(* IEC 61131-3 sources: OpenPLC_Sample_Programs/successed_ST (part 7) *)

(* ---- Scenario7v1_Final.xml_Main.st ---- *)
TYPE
    Magazin_states_t : (Green_Lamp , Init , Interstep , Magazin_Init , Magazin_Init_2 , Slider_Move_Back , Start_Magazin , Step0 , Step1 , convey);
    Stamp_states_t : (Green_Lamp , Init , Interstep , Interstep_2 , StampProcess , StampSliderBack , StampSliderForward , Stamp_Init_1 , Stamp_Init_2 , Stamp_Init_3 , Stamp_Init_4 , Start_Stamp , Step0 , Step1 , Step2);
    Crane_states_t : (Crane_Go_Up , Crane_Init , Crane_Init_2 , Crane_Lift_At_Stamp , Crane_Lift_At_Stamp2 , Crane_Lift_Conveyor , Crane_Lift_Conveyor2 , Crane_Lift_Conveyor_Black , Crane_Lift_Magazin , Crane_Lift_Magazin_Metallic , Crane_Lift_NOT_Metallic_Black , Crane_Lower , Crane_On_Conveyor , Crane_On_Conveyor_Metallic , Crane_On_Conveyor_Metallic2 , Crane_On_Conveyor_Not_Metallica_Black , Crane_On_Stamp_Metallic , Crane_On_Stamp_Metallic2 , Crane_On_Stamp_Metallic2_Lower , Crane_On_Stamp_Stop_Black , Crane_Turn_Left_Back_To_Stamp , Crane_Turn_Left_From_Stamp , Crane_Turn_Left_Metallic , Crane_Turn_Left_Metallic2 , Crane_Turn_Left_NOT_Metallic , Crane_Turn_Left_NOT_Metallic_Black , Crane_Turn_Right_From_Stamp , Init , Interstep , Interstep_2 , Interstep_4 , Lower_Crane , Magazin_Stop , Magazin_Stop_Black , Magazin_Stop_Final , No_Workpiece_ready , Reset_interconnect , Start_Crane , Step0 , Step4 , Suck_At_Stamp , Suck_At_Stamp2 , TimeDelay , Turn_Right , Turn_Right_Black , Turn_Right_Final , pause , release , release2 , release_Black , release_Workpiece);
END_TYPE

FUNCTION_BLOCK Crane_FB
    VAR_INPUT  CraneDown : BOOL; END_VAR
    VAR_OUTPUT  CraneLower : BOOL; END_VAR
    VAR_INPUT  CraneOnConveyor : BOOL; END_VAR
    VAR_INPUT  CraneOnMagazin : BOOL; END_VAR
    VAR_INPUT  CranePositionStamp : BOOL; END_VAR
    VAR_INPUT  CraneSucked : BOOL; END_VAR
    VAR_OUTPUT  CraneTurnClockwise : BOOL; END_VAR
    VAR_OUTPUT  CraneTurnCounterclockwise : BOOL; END_VAR
    VAR_INPUT  CraneUp : BOOL; END_VAR
    VAR  Duration1 : TIME := TIME#1s500ms; END_VAR
    VAR_INPUT  MagazinCapacitiveSensor : BOOL; END_VAR
    VAR_INPUT  MagazinOpticalSensor : BOOL; END_VAR
    VAR_OUTPUT  MagazinVacuumOff : BOOL; END_VAR
    VAR_OUTPUT  MagazinVacuumOn : BOOL; END_VAR
    VAR  SFCInit : BOOL; END_VAR
    VAR_INPUT  SFCReset : BOOL; END_VAR
    VAR_INPUT  SliderMovedOut : BOOL; END_VAR
    VAR_INPUT  SliderNotMovedOut : BOOL; END_VAR
    VAR_INPUT  StampLowered : BOOL; END_VAR
    VAR_INPUT  StampSliderFilled : BOOL; END_VAR
    VAR_INPUT  StampSliderSensorMovedOut : BOOL; END_VAR
    VAR_INPUT  StartButtonMagazin : BOOL; END_VAR
    VAR_OUTPUT  StartCommandCrane : BOOL; END_VAR
    VAR_INPUT  StartVar : BOOL; END_VAR
    VAR  TimeDelay_Timer : TON; END_VAR
    VAR  TimeDelay_Timer_Duration : TIME := TIME#50ms; END_VAR
    VAR  TimeDelay_Timer_interconnect : BOOL; END_VAR
    VAR  Timer1 : TON; END_VAR
    VAR_INPUT  WorkpieceReady : BOOL; END_VAR
    VAR  _state : Crane_states_t; END_VAR
    VAR  _transit : BOOL; END_VAR
    VAR  actualtime1 : TIME; END_VAR
    VAR  interconnect : BOOL; END_VAR
    VAR  interconnectCraneStartCommand : BOOL; END_VAR

    CASE _state OF
        Crane_states_t#Crane_Go_Up:
            _transit := FALSE;
            CraneLower := FALSE;
            IF ((CraneUp AND WorkpieceReady) AND (NOT MagazinCapacitiveSensor AND NOT MagazinOpticalSensor)) THEN
                _transit := TRUE;
                _state := Crane_states_t#Turn_Right_Black;
            ELSIF ((CraneUp AND WorkpieceReady) AND (MagazinCapacitiveSensor OR MagazinOpticalSensor)) THEN
                _transit := TRUE;
                _state := Crane_states_t#pause;
            ELSIF (CraneUp AND NOT WorkpieceReady) THEN
                _transit := TRUE;
                _state := Crane_states_t#Step4;
            END_IF;

        Crane_states_t#Crane_Init:
            _transit := FALSE;
            CraneLower := TRUE;
            interconnectCraneStartCommand := FALSE;
            IF CraneDown THEN
                _transit := TRUE;
                _state := Crane_states_t#Crane_Init_2;
            END_IF;

        Crane_states_t#Crane_Init_2:
            _transit := FALSE;
            CraneLower := FALSE;
            IF CraneUp THEN
                _transit := TRUE;
                _state := Crane_states_t#Interstep;
            END_IF;

        Crane_states_t#Crane_Lift_At_Stamp:
            _transit := FALSE;
            CraneLower := FALSE;
            IF CraneUp THEN
                _transit := TRUE;
                _state := Crane_states_t#Crane_Turn_Left_From_Stamp;
            END_IF;

        Crane_states_t#Crane_Lift_At_Stamp2:
            _transit := FALSE;
            CraneLower := FALSE;
            IF CraneUp THEN
                _transit := TRUE;
                _state := Crane_states_t#Crane_Turn_Right_From_Stamp;
            END_IF;

        Crane_states_t#Crane_Lift_Conveyor:
            _transit := FALSE;
            CraneLower := FALSE;
            IF TRUE THEN
                _transit := TRUE;
                _state := Crane_states_t#Interstep;
            END_IF;

        Crane_states_t#Crane_Lift_Conveyor2:
            _transit := FALSE;
            CraneLower := FALSE;
            IF TRUE THEN
                _transit := TRUE;
                _state := Crane_states_t#Interstep;
            END_IF;

        Crane_states_t#Crane_Lift_Conveyor_Black:
            _transit := FALSE;
            CraneLower := FALSE;
            IF CraneUp THEN
                _transit := TRUE;
                _state := Crane_states_t#Crane_Turn_Left_Back_To_Stamp;
            END_IF;

        Crane_states_t#Crane_Lift_Magazin:
            _transit := FALSE;
            CraneLower := FALSE;
            IF CraneUp THEN
                _transit := TRUE;
                _state := Crane_states_t#Crane_Turn_Left_NOT_Metallic;
            END_IF;

        Crane_states_t#Crane_Lift_Magazin_Metallic:
            _transit := FALSE;
            CraneLower := FALSE;
            IF CraneUp THEN
                _transit := TRUE;
                _state := Crane_states_t#Crane_Turn_Left_Metallic;
            END_IF;

        Crane_states_t#Crane_Lift_NOT_Metallic_Black:
            _transit := FALSE;
            CraneLower := FALSE;
            IF CraneUp THEN
                _transit := TRUE;
                _state := Crane_states_t#Crane_Turn_Left_NOT_Metallic_Black;
            END_IF;

        Crane_states_t#Crane_Lower:
            _transit := FALSE;
            MagazinVacuumOn := TRUE;
            MagazinVacuumOff := FALSE;
            CraneLower := TRUE;
            IF CraneSucked THEN
                _transit := TRUE;
                _state := Crane_states_t#Step0;
            END_IF;

        Crane_states_t#Crane_On_Conveyor:
            _transit := FALSE;
            CraneTurnCounterclockwise := FALSE;
            CraneTurnClockwise := FALSE;
            CraneLower := TRUE;
            IF CraneDown THEN
                _transit := TRUE;
                _state := Crane_states_t#release;
            END_IF;

        Crane_states_t#Crane_On_Conveyor_Metallic:
            _transit := FALSE;
            CraneTurnCounterclockwise := FALSE;
            CraneTurnClockwise := FALSE;
            CraneLower := TRUE;
            IF CraneDown THEN
                _transit := TRUE;
                _state := Crane_states_t#release;
            END_IF;

        Crane_states_t#Crane_On_Conveyor_Metallic2:
            _transit := FALSE;
            CraneTurnCounterclockwise := FALSE;
            CraneTurnClockwise := FALSE;
            CraneLower := TRUE;
            IF CraneDown THEN
                _transit := TRUE;
                _state := Crane_states_t#release2;
            END_IF;

        Crane_states_t#Crane_On_Conveyor_Not_Metallica_Black:
            _transit := FALSE;
            CraneTurnCounterclockwise := FALSE;
            CraneTurnClockwise := FALSE;
            CraneLower := TRUE;
            IF CraneDown THEN
                _transit := TRUE;
                _state := Crane_states_t#release_Black;
            END_IF;

        Crane_states_t#Crane_On_Stamp_Metallic:
            _transit := FALSE;
            CraneTurnCounterclockwise := FALSE;
            CraneTurnClockwise := FALSE;
            CraneLower := TRUE;
            IF CraneDown THEN
                _transit := TRUE;
                _state := Crane_states_t#release_Workpiece;
            END_IF;

        Crane_states_t#Crane_On_Stamp_Metallic2:
            _transit := FALSE;
            CraneTurnCounterclockwise := FALSE;
            CraneTurnClockwise := FALSE;
            IF StampLowered THEN
                _transit := TRUE;
                _state := Crane_states_t#Interstep_4;
            END_IF;

        Crane_states_t#Crane_On_Stamp_Metallic2_Lower:
            _transit := FALSE;
            CraneLower := TRUE;
            IF CraneDown THEN
                _transit := TRUE;
                _state := Crane_states_t#Suck_At_Stamp2;
            END_IF;

        Crane_states_t#Crane_On_Stamp_Stop_Black:
            _transit := FALSE;
            CraneTurnClockwise := FALSE;
            CraneTurnCounterclockwise := FALSE;
            IF TRUE THEN
                _transit := TRUE;
                _state := Crane_states_t#Reset_interconnect;
            END_IF;

        Crane_states_t#Crane_Turn_Left_Back_To_Stamp:
            _transit := FALSE;
            CraneTurnCounterclockwise := TRUE;
            CraneTurnClockwise := FALSE;
            IF CranePositionStamp THEN
                _transit := TRUE;
                _state := Crane_states_t#Crane_On_Stamp_Stop_Black;
            END_IF;

        Crane_states_t#Crane_Turn_Left_From_Stamp:
            _transit := FALSE;
            CraneTurnClockwise := TRUE;
            CraneTurnCounterclockwise := FALSE;
            IF CraneOnConveyor THEN
                _transit := TRUE;
                _state := Crane_states_t#Crane_On_Conveyor_Metallic;
            END_IF;

        Crane_states_t#Crane_Turn_Left_Metallic:
            _transit := FALSE;
            CraneTurnCounterclockwise := TRUE;
            CraneTurnClockwise := FALSE;
            IF CranePositionStamp THEN
                _transit := TRUE;
                _state := Crane_states_t#Crane_On_Stamp_Metallic;
            END_IF;

        Crane_states_t#Crane_Turn_Left_Metallic2:
            _transit := FALSE;
            CraneTurnCounterclockwise := TRUE;
            CraneTurnClockwise := FALSE;
            IF CranePositionStamp THEN
                _transit := TRUE;
                _state := Crane_states_t#Crane_On_Stamp_Metallic2;
            END_IF;

        Crane_states_t#Crane_Turn_Left_NOT_Metallic:
            _transit := FALSE;
            CraneTurnCounterclockwise := TRUE;
            CraneTurnClockwise := FALSE;
            IF CraneOnConveyor THEN
                _transit := TRUE;
                _state := Crane_states_t#Crane_On_Conveyor;
            END_IF;

        Crane_states_t#Crane_Turn_Left_NOT_Metallic_Black:
            _transit := FALSE;
            CraneTurnCounterclockwise := TRUE;
            CraneTurnClockwise := FALSE;
            IF CraneOnConveyor THEN
                _transit := TRUE;
                _state := Crane_states_t#Crane_On_Conveyor_Not_Metallica_Black;
            END_IF;

        Crane_states_t#Crane_Turn_Right_From_Stamp:
            _transit := FALSE;
            CraneTurnClockwise := TRUE;
            CraneTurnCounterclockwise := FALSE;
            IF CraneOnConveyor THEN
                _transit := TRUE;
                _state := Crane_states_t#Crane_On_Conveyor_Metallic2;
            END_IF;

        Crane_states_t#Init:
            _transit := FALSE;
            IF TRUE THEN
                _transit := TRUE;
                _state := Crane_states_t#Start_Crane;
            END_IF;

        Crane_states_t#Interstep:
            _transit := FALSE;
            StartCommandCrane := TRUE;
            IF StartVar THEN
                _transit := TRUE;
                _state := Crane_states_t#Interstep_2;
            END_IF;

        Crane_states_t#Interstep_2:
            _transit := FALSE;
            IF SliderMovedOut THEN
                _transit := TRUE;
                _state := Crane_states_t#TimeDelay;
            END_IF;

        Crane_states_t#Interstep_4:
            _transit := FALSE;
            IF StampSliderSensorMovedOut THEN
                _transit := TRUE;
                _state := Crane_states_t#Crane_On_Stamp_Metallic2_Lower;
            END_IF;

        Crane_states_t#Lower_Crane:
            _transit := FALSE;
            CraneLower := TRUE;
            IF CraneDown THEN
                _transit := TRUE;
                _state := Crane_states_t#Suck_At_Stamp;
            END_IF;

        Crane_states_t#Magazin_Stop:
            _transit := FALSE;
            CraneTurnClockwise := FALSE;
            CraneTurnCounterclockwise := FALSE;
            IF TRUE THEN
                _transit := TRUE;
                _state := Crane_states_t#Crane_Lower;
            END_IF;

        Crane_states_t#Magazin_Stop_Black:
            _transit := FALSE;
            CraneTurnClockwise := FALSE;
            CraneTurnCounterclockwise := FALSE;
            MagazinVacuumOn := TRUE;
            MagazinVacuumOff := FALSE;
            CraneLower := TRUE;
            IF CraneSucked THEN
                _transit := TRUE;
                _state := Crane_states_t#Crane_Lift_NOT_Metallic_Black;
            END_IF;

        Crane_states_t#Magazin_Stop_Final:
            _transit := FALSE;
            CraneTurnClockwise := FALSE;
            CraneTurnCounterclockwise := FALSE;
            IF TRUE THEN
                _transit := TRUE;
                _state := Crane_states_t#Start_Crane;
            END_IF;

        Crane_states_t#No_Workpiece_ready:
            _transit := FALSE;
            MagazinVacuumOn := FALSE;
            MagazinVacuumOff := FALSE;
            CraneLower := FALSE;
            IF NOT StampSliderFilled THEN
                _transit := TRUE;
                _state := Crane_states_t#Turn_Right_Final;
            ELSIF StampSliderFilled THEN
                _transit := TRUE;
                _state := Crane_states_t#Crane_Turn_Left_Metallic2;
            END_IF;

        Crane_states_t#Reset_interconnect:
            _transit := FALSE;
            interconnect := FALSE;
            Timer1(IN := FALSE, PT := TIME#1ms);
            IF SliderMovedOut THEN
                _transit := TRUE;
                _state := Crane_states_t#Lower_Crane;
            END_IF;

        Crane_states_t#Start_Crane:
            _transit := FALSE;
            CraneLower := FALSE;
            MagazinVacuumOff := FALSE;
            MagazinVacuumOn := FALSE;
            CraneTurnCounterclockwise := FALSE;
            CraneTurnClockwise := FALSE;
            StartVar := FALSE;
            StartCommandCrane := FALSE;
            IF (StartButtonMagazin = TRUE) THEN
                interconnectCraneStartCommand := TRUE;
            END_IF;
            IF interconnectCraneStartCommand THEN
                _transit := TRUE;
                _state := Crane_states_t#Crane_Init;
            END_IF;

        Crane_states_t#Step0:
            _transit := FALSE;
            IF (MagazinCapacitiveSensor OR MagazinOpticalSensor) THEN
                _transit := TRUE;
                _state := Crane_states_t#Crane_Lift_Magazin_Metallic;
            ELSIF (NOT MagazinCapacitiveSensor AND NOT MagazinOpticalSensor) THEN
                _transit := TRUE;
                _state := Crane_states_t#Crane_Lift_Magazin;
            END_IF;

        Crane_states_t#Step4:
            _transit := FALSE;
            IF TRUE THEN
                _transit := TRUE;
                _state := Crane_states_t#Interstep;
            END_IF;

        Crane_states_t#Suck_At_Stamp:
            _transit := FALSE;
            MagazinVacuumOn := TRUE;
            MagazinVacuumOff := FALSE;
            IF CraneSucked THEN
                _transit := TRUE;
                _state := Crane_states_t#Crane_Lift_At_Stamp;
            END_IF;

        Crane_states_t#Suck_At_Stamp2:
            _transit := FALSE;
            MagazinVacuumOn := TRUE;
            MagazinVacuumOff := FALSE;
            IF CraneSucked THEN
                _transit := TRUE;
                _state := Crane_states_t#Crane_Lift_At_Stamp2;
            END_IF;

        Crane_states_t#TimeDelay:
            _transit := FALSE;
            TimeDelay_Timer(IN := TRUE, PT := TimeDelay_Timer_Duration);
            TimeDelay_Timer_interconnect := TimeDelay_Timer.Q;
            IF (WorkpieceReady AND TimeDelay_Timer_interconnect) THEN
                _transit := TRUE;
                _state := Crane_states_t#Turn_Right;
            ELSIF (NOT WorkpieceReady AND TimeDelay_Timer_interconnect) THEN
                _transit := TRUE;
                _state := Crane_states_t#No_Workpiece_ready;
            END_IF;

        Crane_states_t#Turn_Right:
            _transit := FALSE;
            CraneTurnClockwise := TRUE;
            CraneTurnCounterclockwise := FALSE;
            IF CraneOnMagazin THEN
                _transit := TRUE;
                _state := Crane_states_t#Magazin_Stop;
            END_IF;

        Crane_states_t#Turn_Right_Black:
            _transit := FALSE;
            CraneTurnClockwise := TRUE;
            CraneTurnCounterclockwise := FALSE;
            IF CraneOnMagazin THEN
                _transit := TRUE;
                _state := Crane_states_t#Magazin_Stop_Black;
            END_IF;

        Crane_states_t#Turn_Right_Final:
            _transit := FALSE;
            CraneTurnClockwise := TRUE;
            CraneTurnCounterclockwise := FALSE;
            IF CraneOnMagazin THEN
                _transit := TRUE;
                _state := Crane_states_t#Magazin_Stop_Final;
            END_IF;

        Crane_states_t#pause:
            _transit := FALSE;
            Timer1(IN := CraneUp, PT := Duration1);
            interconnect := Timer1.Q;
            IF interconnect THEN
                _transit := TRUE;
                _state := Crane_states_t#Reset_interconnect;
            END_IF;

        Crane_states_t#release:
            _transit := FALSE;
            MagazinVacuumOff := TRUE;
            MagazinVacuumOn := FALSE;
            IF TRUE THEN
                _transit := TRUE;
                _state := Crane_states_t#Crane_Lift_Conveyor;
            END_IF;

        Crane_states_t#release2:
            _transit := FALSE;
            MagazinVacuumOff := TRUE;
            MagazinVacuumOn := FALSE;
            IF TRUE THEN
                _transit := TRUE;
                _state := Crane_states_t#Crane_Lift_Conveyor2;
            END_IF;

        Crane_states_t#release_Black:
            _transit := FALSE;
            MagazinVacuumOn := FALSE;
            MagazinVacuumOff := TRUE;
            IF TRUE THEN
                _transit := TRUE;
                _state := Crane_states_t#Crane_Lift_Conveyor_Black;
            END_IF;

        Crane_states_t#release_Workpiece:
            _transit := FALSE;
            MagazinVacuumOff := TRUE;
            MagazinVacuumOn := FALSE;
            IF TRUE THEN
                _transit := TRUE;
                _state := Crane_states_t#Crane_Go_Up;
            END_IF;

            END_CASE;
END_FUNCTION_BLOCK

FUNCTION_BLOCK Magazin
    VAR CraneDown : BOOL; END_VAR
    VAR CraneLower : BOOL; END_VAR
    VAR CraneOnConveyor : BOOL; END_VAR
    VAR CraneOnMagazin : BOOL; END_VAR
    VAR CraneSucked : BOOL; END_VAR
    VAR CraneTurnClockwise : BOOL; END_VAR
    VAR CraneTurnCounterclockwise : BOOL; END_VAR
    VAR CraneUp : BOOL; END_VAR
    VAR MagazinGreenLamp : BOOL; END_VAR
    VAR MagazinSlider : BOOL; END_VAR
    VAR MagazinVacuumOff : BOOL; END_VAR
    VAR MagazinVacuumOn : BOOL; END_VAR
    VAR MagazinWhiteLamp : BOOL; END_VAR
    VAR SFCInit : BOOL; END_VAR
    VAR SFCReset : BOOL; END_VAR
    VAR SliderMovedOut : BOOL; END_VAR
    VAR SliderNotMovedOut : BOOL; END_VAR
    VAR StartButtonMagazin : BOOL; END_VAR
    VAR StartCommandMagazin : BOOL; END_VAR
    VAR StartVar : BOOL; END_VAR
    VAR WorkpieceReady : BOOL; END_VAR
    VAR _state : Magazin_states_t; END_VAR
    VAR _transit : BOOL; END_VAR
    VAR interconnectMagazinStartCommand : BOOL; END_VAR

    CASE _state OF
        Magazin_states_t#Green_Lamp:
            _transit := FALSE;
            MagazinGreenLamp := TRUE;
            interconnectMagazinStartCommand := FALSE;
            IF TRUE THEN
                _transit := TRUE;
                _state := Magazin_states_t#Magazin_Init;
            END_IF;

        Magazin_states_t#Init:
            _transit := FALSE;
            IF TRUE THEN
                _transit := TRUE;
                _state := Magazin_states_t#Start_Magazin;
            END_IF;

        Magazin_states_t#Interstep:
            _transit := FALSE;
            StartCommandMagazin := TRUE;
            IF StartVar THEN
                _transit := TRUE;
                _state := Magazin_states_t#convey;
            END_IF;

        Magazin_states_t#Magazin_Init:
            _transit := FALSE;
            MagazinSlider := TRUE;
            IF TRUE THEN
                _transit := TRUE;
                _state := Magazin_states_t#Magazin_Init_2;
            END_IF;

        Magazin_states_t#Magazin_Init_2:
            _transit := FALSE;
            MagazinSlider := FALSE;
            IF TRUE THEN
                _transit := TRUE;
                _state := Magazin_states_t#Interstep;
            END_IF;

        Magazin_states_t#Slider_Move_Back:
            _transit := FALSE;
            IF ((SliderMovedOut = TRUE) AND (SliderNotMovedOut = FALSE)) THEN
                MagazinSlider := FALSE;
            END_IF;
            IF CraneUp THEN
                _transit := TRUE;
                _state := Magazin_states_t#Step1;
            END_IF;

        Magazin_states_t#Start_Magazin:
            _transit := FALSE;
            MagazinSlider := FALSE;
            MagazinGreenLamp := FALSE;
            StartVar := FALSE;
            StartCommandMagazin := FALSE;
            IF (StartButtonMagazin = TRUE) THEN
                interconnectMagazinStartCommand := TRUE;
            END_IF;
            IF interconnectMagazinStartCommand THEN
                _transit := TRUE;
                _state := Magazin_states_t#Green_Lamp;
            END_IF;

        Magazin_states_t#Step0:
            _transit := FALSE;
            IF CraneDown THEN
                _transit := TRUE;
                _state := Magazin_states_t#Slider_Move_Back;
            END_IF;

        Magazin_states_t#Step1:
            _transit := FALSE;
            IF CraneOnConveyor THEN
                _transit := TRUE;
                _state := Magazin_states_t#Interstep;
            END_IF;

        Magazin_states_t#convey:
            _transit := FALSE;
            IF SliderNotMovedOut THEN
                MagazinSlider := TRUE;
            END_IF;
            IF CraneOnMagazin THEN
                _transit := TRUE;
                _state := Magazin_states_t#Step0;
            END_IF;

            END_CASE;
END_FUNCTION_BLOCK

FUNCTION_BLOCK Stamp_FB
    VAR_INPUT  CraneDown : BOOL; END_VAR
    VAR_INPUT  CraneOnConveyor : BOOL; END_VAR
    VAR_INPUT  CranePositionStamp : BOOL; END_VAR
    VAR_INPUT  CraneSucked : BOOL; END_VAR
    VAR_INPUT  CraneUp : BOOL; END_VAR
    VAR  Duration : TIME := TIME#500.0ms; END_VAR
    VAR  SFCInit : BOOL; END_VAR
    VAR_INPUT  SFCReset : BOOL; END_VAR
    VAR_OUTPUT  StampGreenLamp : BOOL; END_VAR
    VAR_INPUT  StampLowered : BOOL; END_VAR
    VAR_OUTPUT  StampPressure : BOOL; END_VAR
    VAR_OUTPUT  StampPusher : BOOL; END_VAR
    VAR_INPUT  StampSliderFilled : BOOL; END_VAR
    VAR_OUTPUT  StampSliderMovedIn : BOOL; END_VAR
    VAR_OUTPUT  StampSliderMovedOut : BOOL; END_VAR
    VAR_INPUT  StampSliderSensorMovedIn : BOOL; END_VAR
    VAR_INPUT  StampSliderSensorMovedOut : BOOL; END_VAR
    VAR_INPUT  StampStartButton : BOOL; END_VAR
    VAR_INPUT  StampUp : BOOL; END_VAR
    VAR_OUTPUT  StampWhiteLamp : BOOL; END_VAR
    VAR_OUTPUT  StartCommandStamp : BOOL; END_VAR
    VAR_INPUT  StartVar : BOOL; END_VAR
    VAR  Timer : TON; END_VAR
    VAR  _state : Stamp_states_t; END_VAR
    VAR  _transit : BOOL; END_VAR
    VAR  interconnect : BOOL; END_VAR
    VAR  interconnectStampStartCommand : BOOL; END_VAR

    CASE _state OF
        Stamp_states_t#Green_Lamp:
            _transit := FALSE;
            StampGreenLamp := TRUE;
            interconnectStampStartCommand := FALSE;
            IF TRUE THEN
                _transit := TRUE;
                _state := Stamp_states_t#Stamp_Init_1;
            END_IF;

        Stamp_states_t#Init:
            _transit := FALSE;
            IF TRUE THEN
                _transit := TRUE;
                _state := Stamp_states_t#Start_Stamp;
            END_IF;

        Stamp_states_t#Interstep:
            _transit := FALSE;
            StartCommandStamp := TRUE;
            IF StartVar THEN
                _transit := TRUE;
                _state := Stamp_states_t#Interstep_2;
            END_IF;

        Stamp_states_t#Interstep_2:
            _transit := FALSE;
            IF StampSliderFilled THEN
                _transit := TRUE;
                _state := Stamp_states_t#Step0;
            END_IF;

        Stamp_states_t#StampProcess:
            _transit := FALSE;
            StampSliderMovedIn := FALSE;
            StampPusher := TRUE;
            IF StampLowered THEN
                _transit := TRUE;
                _state := Stamp_states_t#Step1;
            END_IF;

        Stamp_states_t#StampSliderBack:
            _transit := FALSE;
            StampSliderMovedIn := TRUE;
            StampSliderMovedOut := FALSE;
            IF StampSliderSensorMovedIn THEN
                _transit := TRUE;
                _state := Stamp_states_t#StampProcess;
            END_IF;

        Stamp_states_t#StampSliderForward:
            _transit := FALSE;
            StampPusher := FALSE;
            StampSliderMovedOut := TRUE;
            IF ((StampLowered = FALSE) AND (StampUp = TRUE)) THEN
                interconnect := FALSE;
            END_IF;
            Timer(IN := FALSE, PT := TIME#1ms);
            IF StampSliderMovedOut THEN
                _transit := TRUE;
                _state := Stamp_states_t#Step2;
            END_IF;

        Stamp_states_t#Stamp_Init_1:
            _transit := FALSE;
            StampSliderMovedIn := TRUE;
            StampSliderMovedOut := FALSE;
            IF StampSliderSensorMovedIn THEN
                _transit := TRUE;
                _state := Stamp_states_t#Stamp_Init_2;
            END_IF;

        Stamp_states_t#Stamp_Init_2:
            _transit := FALSE;
            StampSliderMovedIn := FALSE;
            StampSliderMovedOut := TRUE;
            IF StampSliderSensorMovedOut THEN
                _transit := TRUE;
                _state := Stamp_states_t#Stamp_Init_3;
            END_IF;

        Stamp_states_t#Stamp_Init_3:
            _transit := FALSE;
            StampPusher := TRUE;
            IF StampLowered THEN
                _transit := TRUE;
                _state := Stamp_states_t#Stamp_Init_4;
            END_IF;

        Stamp_states_t#Stamp_Init_4:
            _transit := FALSE;
            StampPusher := FALSE;
            IF StampUp THEN
                _transit := TRUE;
                _state := Stamp_states_t#Interstep;
            END_IF;

        Stamp_states_t#Start_Stamp:
            _transit := FALSE;
            StampSliderMovedOut := FALSE;
            StampSliderMovedIn := FALSE;
            StampPusher := FALSE;
            StampGreenLamp := FALSE;
            StampPressure := FALSE;
            StartCommandStamp := FALSE;
            IF (StampStartButton = TRUE) THEN
                interconnectStampStartCommand := TRUE;
            END_IF;
            IF interconnectStampStartCommand THEN
                _transit := TRUE;
                _state := Stamp_states_t#Green_Lamp;
            END_IF;

        Stamp_states_t#Step0:
            _transit := FALSE;
            IF CraneUp THEN
                _transit := TRUE;
                _state := Stamp_states_t#StampSliderBack;
            END_IF;

        Stamp_states_t#Step1:
            _transit := FALSE;
            Timer(IN := StampLowered, PT := TIME#12ms);
            interconnect := Timer.Q;
            IF interconnect THEN
                _transit := TRUE;
                _state := Stamp_states_t#StampSliderForward;
            END_IF;

        Stamp_states_t#Step2:
            _transit := FALSE;
            IF (CraneOnConveyor AND NOT StampSliderFilled) THEN
                _transit := TRUE;
                _state := Stamp_states_t#Interstep;
            END_IF;

            END_CASE;
END_FUNCTION_BLOCK

PROGRAM MAIN

VAR  ACTUATOR_ANALOGCRANEPRESSURE : INT; END_VAR
VAR  ACTUATOR_CRANELOWER : BOOL; END_VAR
VAR  ACTUATOR_CRANETURNCLOCKWISE : BOOL; END_VAR
VAR  ACTUATOR_CRANETURNCOUNTERCLOCKWISE : BOOL; END_VAR
VAR  ACTUATOR_MAGAZINGREENLAMP : BOOL; END_VAR
VAR  ACTUATOR_MAGAZINSLIDER : BOOL; END_VAR
VAR  ACTUATOR_MAGAZINVACUUMOFF : BOOL; END_VAR
VAR  ACTUATOR_MAGAZINVACUUMON : BOOL; END_VAR
VAR  ACTUATOR_MAGAZINWHITELAMP : BOOL; END_VAR
VAR  ACTUATOR_STAMPGREENLAMP : BOOL; END_VAR
VAR  ACTUATOR_STAMPPUSHER : BOOL; END_VAR
VAR  ACTUATOR_STAMPSLIDERMOVEDIN : BOOL; END_VAR
VAR  ACTUATOR_STAMPSLIDERMOVEDOUT : BOOL; END_VAR
VAR  ACTUATOR_STAMPWHITELAMP : BOOL; END_VAR
VAR  CRANE : CRANE_FB; END_VAR
VAR  MAG : MAGAZIN; END_VAR
VAR  SENSOR_CRANEDOWN : BOOL; END_VAR
VAR  SENSOR_CRANEONCONVEYOR : BOOL; END_VAR
VAR  SENSOR_CRANEONMAGAZIN : BOOL; END_VAR
VAR  SENSOR_CRANEPOSITION : BOOL; END_VAR
VAR  SENSOR_CRANEPOSITIONSTAMP : BOOL; END_VAR
VAR  SENSOR_CRANESUCKED : BOOL; END_VAR
VAR  SENSOR_CRANEUP : BOOL; END_VAR
VAR  SENSOR_MAGAZINCAPACITIVESENSOR : BOOL; END_VAR
VAR  SENSOR_MAGAZINEMERGENCYSTOP : BOOL; END_VAR
VAR  SENSOR_MAGAZINOPTICALSENSOR : BOOL; END_VAR
VAR  SENSOR_MAGAZINSWITCHMANUELLAUTOMATIC : BOOL; END_VAR
VAR  SENSOR_SLIDERMOVEDOUT : BOOL; END_VAR
VAR  SENSOR_SLIDERNOTMOVEDOUT : BOOL; END_VAR
VAR  SENSOR_STAMPEMERGENCYSTOP : BOOL; END_VAR
VAR  SENSOR_STAMPLOWERED : BOOL; END_VAR
VAR  SENSOR_STAMPSLIDERFILLED : BOOL; END_VAR
VAR  SENSOR_STAMPSLIDERSENSORMOVEDIN : BOOL; END_VAR
VAR  SENSOR_STAMPSLIDERSENSORMOVEDOUT : BOOL; END_VAR
VAR  SENSOR_STAMPSTARTBUTTON : BOOL; END_VAR
VAR  SENSOR_STAMPSWITCHMANUELLAUTOMATIC : BOOL; END_VAR
VAR  SENSOR_STAMPUP : BOOL; END_VAR
VAR  SENSOR_STARTBUTTONMAGAZIN : BOOL; END_VAR
VAR  SENSOR_WORKPIECEREADY : BOOL; END_VAR
VAR  STAMP : STAMP_FB; END_VAR
MAG.SLIDERNOTMOVEDOUT := SENSOR_SLIDERNOTMOVEDOUT;
MAG.SLIDERMOVEDOUT := SENSOR_SLIDERMOVEDOUT;
MAG.CRANEONMAGAZIN := SENSOR_CRANEONMAGAZIN;
MAG.CRANEDOWN := SENSOR_CRANEDOWN;
MAG.CRANEUP := SENSOR_CRANEUP;
MAG.CRANEONCONVEYOR := SENSOR_CRANEONCONVEYOR;
MAG.WORKPIECEREADY := SENSOR_WORKPIECEREADY;
MAG.STARTBUTTONMAGAZIN := SENSOR_STARTBUTTONMAGAZIN;
ACTUATOR_MAGAZINSLIDER := MAG.MAGAZINSLIDER;
ACTUATOR_MAGAZINGREENLAMP := MAG.MAGAZINGREENLAMP;
CRANE.CRANEUP := SENSOR_CRANEUP;
CRANE.CRANEONCONVEYOR := SENSOR_CRANEONCONVEYOR;
CRANE.CRANEDOWN := SENSOR_CRANEDOWN;
CRANE.CRANESUCKED := SENSOR_CRANESUCKED;
CRANE.CRANEONMAGAZIN := SENSOR_CRANEONMAGAZIN;
CRANE.MAGAZINCAPACITIVESENSOR := SENSOR_MAGAZINCAPACITIVESENSOR;
CRANE.CRANEPOSITIONSTAMP := SENSOR_CRANEPOSITIONSTAMP;
CRANE.SLIDERMOVEDOUT := SENSOR_SLIDERMOVEDOUT;
CRANE.WORKPIECEREADY := SENSOR_WORKPIECEREADY;
CRANE.MAGAZINOPTICALSENSOR := SENSOR_MAGAZINOPTICALSENSOR;
CRANE.STAMPSLIDERFILLED := SENSOR_STAMPSLIDERFILLED;
CRANE.STAMPSLIDERSENSORMOVEDOUT := SENSOR_STAMPSLIDERSENSORMOVEDOUT;
CRANE.STAMPLOWERED := SENSOR_STAMPLOWERED;
CRANE.STARTBUTTONMAGAZIN := SENSOR_STARTBUTTONMAGAZIN;
ACTUATOR_CRANETURNCOUNTERCLOCKWISE := CRANE.CRANETURNCOUNTERCLOCKWISE;
ACTUATOR_CRANETURNCLOCKWISE := CRANE.CRANETURNCLOCKWISE;
ACTUATOR_CRANELOWER := CRANE.CRANELOWER;
ACTUATOR_MAGAZINVACUUMOFF := CRANE.MAGAZINVACUUMOFF;
ACTUATOR_MAGAZINVACUUMON := CRANE.MAGAZINVACUUMON;
STAMP.STAMPSLIDERSENSORMOVEDOUT := SENSOR_STAMPSLIDERSENSORMOVEDOUT;
STAMP.STAMPSLIDERSENSORMOVEDIN := SENSOR_STAMPSLIDERSENSORMOVEDIN;
STAMP.STAMPSLIDERFILLED := SENSOR_STAMPSLIDERFILLED;
STAMP.STAMPUP := SENSOR_STAMPUP;
STAMP.STAMPLOWERED := SENSOR_STAMPLOWERED;
STAMP.CRANEDOWN := SENSOR_CRANEDOWN;
STAMP.CRANEUP := SENSOR_CRANEUP;
STAMP.CRANESUCKED := SENSOR_CRANESUCKED;
STAMP.CRANEPOSITIONSTAMP := SENSOR_CRANEPOSITIONSTAMP;
STAMP.CRANEONCONVEYOR := SENSOR_CRANEONCONVEYOR;
STAMP.STAMPSTARTBUTTON := SENSOR_STAMPSTARTBUTTON;
ACTUATOR_STAMPSLIDERMOVEDOUT := STAMP.STAMPSLIDERMOVEDOUT;
ACTUATOR_STAMPSLIDERMOVEDIN := STAMP.STAMPSLIDERMOVEDIN;
ACTUATOR_STAMPWHITELAMP := STAMP.STAMPWHITELAMP;
ACTUATOR_STAMPPUSHER := STAMP.STAMPPUSHER;
ACTUATOR_STAMPGREENLAMP := STAMP.STAMPGREENLAMP;
ACTUATOR_ANALOGCRANEPRESSURE := INT#6000;
IF (SENSOR_STAMPEMERGENCYSTOP AND SENSOR_MAGAZINEMERGENCYSTOP) THEN
    MAG();
    CRANE();
    STAMP();
    IF (ACTUATOR_MAGAZINGREENLAMP AND ACTUATOR_STAMPGREENLAMP) THEN
        IF ((STAMP.STARTCOMMANDSTAMP AND CRANE.STARTCOMMANDCRANE) AND MAG.STARTCOMMANDMAGAZIN) THEN
            CRANE.STARTVAR := TRUE;
            MAG.STARTVAR := TRUE;
            STAMP.STARTVAR := TRUE;
        END_IF;
    END_IF;
    CRANE.SFCRESET := FALSE;
    MAG.SFCRESET := FALSE;
    STAMP.SFCRESET := FALSE;
ELSIF (NOT SENSOR_STAMPEMERGENCYSTOP OR NOT SENSOR_MAGAZINEMERGENCYSTOP) THEN
    ACTUATOR_MAGAZINSLIDER := FALSE;
    ACTUATOR_CRANELOWER := FALSE;
    ACTUATOR_MAGAZINVACUUMON := FALSE;
    ACTUATOR_MAGAZINVACUUMOFF := TRUE;
    ACTUATOR_MAGAZINGREENLAMP := FALSE;
    ACTUATOR_CRANETURNCOUNTERCLOCKWISE := FALSE;
    ACTUATOR_CRANETURNCLOCKWISE := FALSE;
    ACTUATOR_STAMPSLIDERMOVEDOUT := TRUE;
    ACTUATOR_STAMPSLIDERMOVEDIN := FALSE;
    ACTUATOR_STAMPGREENLAMP := FALSE;
    ACTUATOR_STAMPPUSHER := FALSE;
    ACTUATOR_ANALOGCRANEPRESSURE := INT#0;
    CRANE.SFCRESET := TRUE;
    MAG.SFCRESET := TRUE;
    STAMP.SFCRESET := TRUE;
    CRANE.STARTVAR := FALSE;
    MAG.STARTVAR := FALSE;
    STAMP.STARTVAR := FALSE;
END_IF;
END_PROGRAM

CONFIGURATION Config0
  RESOURCE Res0 ON PLC
    TASK TASK0(INTERVAL := T#50MS, PRIORITY := 0);
    PROGRAM INSTANCE0 WITH TASK0 : MAIN;
  END_RESOURCE
END_CONFIGURATION

(* ---- Scenario8_Final.xml.st ---- *)
TYPE
    MAGAZIN_STATES_T : (GREEN_LAMP , INIT , INTERSTEP , MAGAZIN_INIT , MAGAZIN_INIT_2 , SLIDER_MOVE_BACK , START_MAGAZIN , STEP0 , STEP1 , CONVEY);
    STAMP_STATES_T : (GREEN_LAMP , INIT , INTERSTEP , INTERSTEP_2 , STAMPPROCESS , STAMPSLIDERBACK , STAMPSLIDERFORWARD , STAMP_INIT_1 , STAMP_INIT_2 , STAMP_INIT_3 , STAMP_INIT_4 , START_STAMP , STEP0 , STEP1 , STEP2);
    CRANE_STATES_T : (CRANE_GO_UP , CRANE_GO_UP_WHITE , CRANE_INIT , CRANE_INIT_2 , CRANE_LIFT_AT_STAMP , CRANE_LIFT_AT_STAMP2 , CRANE_LIFT_CONVEYOR , CRANE_LIFT_CONVEYOR2 , CRANE_LIFT_CONVEYOR_BLACK , CRANE_LIFT_MAGAZIN , CRANE_LIFT_MAGAZIN_METALLIC , CRANE_LIFT_MAGAZINE_WHITE , CRANE_LIFT_NOT_METALLIC_BLACK , CRANE_LOWER , CRANE_ON_CONVEYOR , CRANE_ON_CONVEYOR_METALLIC , CRANE_ON_CONVEYOR_METALLIC2 , CRANE_ON_CONVEYOR_NOT_METALLICA_BLACK , CRANE_ON_STAMP_METALLIC , CRANE_ON_STAMP_METALLIC2 , CRANE_ON_STAMP_METALLIC2_LOWER , CRANE_ON_STAMP_STOP_BLACK , CRANE_ON_STAMP_WHITE , CRANE_TURN_LEFT_BACK_TO_STAMP , CRANE_TURN_LEFT_FROM_STAMP , CRANE_TURN_LEFT_METALLIC , CRANE_TURN_LEFT_METALLIC2 , CRANE_TURN_LEFT_NOT_METALLIC , CRANE_TURN_LEFT_NOT_METALLIC_BLACK , CRANE_TURN_LEFT_WHITE , CRANE_TURN_RIGHT_FROM_STAMP , INIT , INTERSTEP , INTERSTEP_2 , INTERSTEP_3 , INTERSTEP_4 , LOWER_CRANE , MAGAZIN_STOP , MAGAZIN_STOP_BLACK , MAGAZIN_STOP_FINAL , NO_WORKPIECE_READY , RESET_INTERCONNECT , STAMP_PRESSURE_PROFILE_SET_METALLIC , STAMP_PRESSURE_PROFILE_SET_WHITE , START_CRANE , STEP0 , STEP2 , STEP3 , STEP4 , SUCK_AT_STAMP , SUCK_AT_STAMP2 , TIMEDELAY , TURN_RIGHT , TURN_RIGHT_BLACK , TURN_RIGHT_FINAL , PAUSE , RELEASE , RELEASE2 , RELEASE_BLACK , RELEASE_WORKPIECE , RELEASE_WORKPIECE_WHITE);
END_TYPE

FUNCTION_BLOCK MAGAZIN
    VAR_INPUT  CRANEDOWN : BOOL; END_VAR
    VAR_OUTPUT  CRANELOWER : BOOL; END_VAR
    VAR_INPUT  CRANEONCONVEYOR : BOOL; END_VAR
    VAR_INPUT  CRANEONMAGAZIN : BOOL; END_VAR
    VAR_INPUT  CRANESUCKED : BOOL; END_VAR
    VAR_OUTPUT  CRANETURNCLOCKWISE : BOOL; END_VAR
    VAR_OUTPUT  CRANETURNCOUNTERCLOCKWISE : BOOL; END_VAR
    VAR_INPUT  CRANEUP : BOOL; END_VAR
    VAR_OUTPUT  MAGAZINGREENLAMP : BOOL; END_VAR
    VAR_OUTPUT  MAGAZINSLIDER : BOOL; END_VAR
    VAR_OUTPUT  MAGAZINVACUUMOFF : BOOL; END_VAR
    VAR_OUTPUT  MAGAZINVACUUMON : BOOL; END_VAR
    VAR_OUTPUT  MAGAZINWHITELAMP : BOOL; END_VAR
    VAR  SFCINIT : BOOL; END_VAR
    VAR_INPUT  SFCRESET : BOOL; END_VAR
    VAR_INPUT  SLIDERMOVEDOUT : BOOL; END_VAR
    VAR_INPUT  SLIDERNOTMOVEDOUT : BOOL; END_VAR
    VAR_INPUT  STARTBUTTONMAGAZIN : BOOL; END_VAR
    VAR_OUTPUT  STARTCOMMANDMAGAZIN : BOOL; END_VAR
    VAR_INPUT  STARTVAR : BOOL; END_VAR
    VAR_INPUT  WORKPIECEREADY : BOOL; END_VAR
    VAR  _STATE : MAGAZIN_STATES_T; END_VAR
    VAR  _TRANSIT : BOOL; END_VAR
    VAR  INTERCONNECTMAGAZINSTARTCOMMAND : BOOL; END_VAR

    CASE _STATE OF
        MAGAZIN_STATES_T#GREEN_LAMP:
            _TRANSIT := FALSE;
            MAGAZINGREENLAMP := TRUE;
            INTERCONNECTMAGAZINSTARTCOMMAND := FALSE;
            IF TRUE THEN
                _TRANSIT := TRUE;
                _STATE := MAGAZIN_STATES_T#MAGAZIN_INIT;
            END_IF;

        MAGAZIN_STATES_T#INIT:
            _TRANSIT := FALSE;
            IF TRUE THEN
                _TRANSIT := TRUE;
                _STATE := MAGAZIN_STATES_T#START_MAGAZIN;
            END_IF;

        MAGAZIN_STATES_T#INTERSTEP:
            _TRANSIT := FALSE;
            STARTCOMMANDMAGAZIN := TRUE;
            IF STARTVAR THEN
                _TRANSIT := TRUE;
                _STATE := MAGAZIN_STATES_T#CONVEY;
            END_IF;

        MAGAZIN_STATES_T#MAGAZIN_INIT:
            _TRANSIT := FALSE;
            MAGAZINSLIDER := TRUE;
            IF TRUE THEN
                _TRANSIT := TRUE;
                _STATE := MAGAZIN_STATES_T#MAGAZIN_INIT_2;
            END_IF;

        MAGAZIN_STATES_T#MAGAZIN_INIT_2:
            _TRANSIT := FALSE;
            MAGAZINSLIDER := FALSE;
            IF TRUE THEN
                _TRANSIT := TRUE;
                _STATE := MAGAZIN_STATES_T#INTERSTEP;
            END_IF;

        MAGAZIN_STATES_T#SLIDER_MOVE_BACK:
            _TRANSIT := FALSE;
            IF ((SLIDERMOVEDOUT = TRUE) AND (SLIDERNOTMOVEDOUT = FALSE)) THEN
                MAGAZINSLIDER := FALSE;
            END_IF;
            IF CRANEUP THEN
                _TRANSIT := TRUE;
                _STATE := MAGAZIN_STATES_T#STEP1;
            END_IF;

        MAGAZIN_STATES_T#START_MAGAZIN:
            _TRANSIT := FALSE;
            MAGAZINSLIDER := FALSE;
            MAGAZINGREENLAMP := FALSE;
            STARTVAR := FALSE;
            STARTCOMMANDMAGAZIN := FALSE;
            IF (STARTBUTTONMAGAZIN = TRUE) THEN
                INTERCONNECTMAGAZINSTARTCOMMAND := TRUE;
            END_IF;
            IF INTERCONNECTMAGAZINSTARTCOMMAND THEN
                _TRANSIT := TRUE;
                _STATE := MAGAZIN_STATES_T#GREEN_LAMP;
            END_IF;

        MAGAZIN_STATES_T#STEP0:
            _TRANSIT := FALSE;
            IF CRANEDOWN THEN
                _TRANSIT := TRUE;
                _STATE := MAGAZIN_STATES_T#SLIDER_MOVE_BACK;
            END_IF;

        MAGAZIN_STATES_T#STEP1:
            _TRANSIT := FALSE;
            IF CRANEONCONVEYOR THEN
                _TRANSIT := TRUE;
                _STATE := MAGAZIN_STATES_T#INTERSTEP;
            END_IF;

        MAGAZIN_STATES_T#CONVEY:
            _TRANSIT := FALSE;
            IF SLIDERNOTMOVEDOUT THEN
                MAGAZINSLIDER := TRUE;
            END_IF;
            IF CRANEONMAGAZIN THEN
                _TRANSIT := TRUE;
                _STATE := MAGAZIN_STATES_T#STEP0;
            END_IF;

            END_CASE;
END_FUNCTION_BLOCK

FUNCTION_BLOCK STAMP_FB
VAR_INPUT  CRANEDOWN : BOOL; END_VAR
VAR_INPUT  CRANEONCONVEYOR : BOOL; END_VAR
VAR_INPUT  CRANEPOSITIONSTAMP : BOOL; END_VAR
VAR_INPUT  CRANESUCKED : BOOL; END_VAR
VAR_INPUT  CRANEUP : BOOL; END_VAR
VAR  DURATION : TIME := TIME#500MS; END_VAR
VAR  SFCINIT : BOOL; END_VAR
VAR_INPUT  SFCRESET : BOOL; END_VAR
VAR_OUTPUT  STAMPGREENLAMP : BOOL; END_VAR
VAR_INPUT  STAMPLOWERED : BOOL; END_VAR
VAR_OUTPUT  STAMPPRESSURE : BOOL; END_VAR
VAR_OUTPUT  STAMPPUSHER : BOOL; END_VAR
VAR_INPUT  STAMPSLIDERFILLED : BOOL; END_VAR
VAR_OUTPUT  STAMPSLIDERMOVEDIN : BOOL; END_VAR
VAR_OUTPUT  STAMPSLIDERMOVEDOUT : BOOL; END_VAR
VAR_INPUT  STAMPSLIDERSENSORMOVEDIN : BOOL; END_VAR
VAR_INPUT  STAMPSLIDERSENSORMOVEDOUT : BOOL; END_VAR
VAR_INPUT  STAMPSTARTBUTTON : BOOL; END_VAR
VAR_INPUT  STAMPUP : BOOL; END_VAR
VAR_OUTPUT  STAMPWHITELAMP : BOOL; END_VAR
VAR_OUTPUT  STARTCOMMANDSTAMP : BOOL; END_VAR
VAR_INPUT  STARTVAR : BOOL; END_VAR
VAR  TIMER : TON; END_VAR
VAR  _STATE : STAMP_STATES_T; END_VAR
VAR  _TRANSIT : BOOL; END_VAR
VAR  INTERCONNECT : BOOL; END_VAR
VAR  INTERCONNECTSTAMPSTARTCOMMAND : BOOL; END_VAR

CASE _STATE OF
    STAMP_STATES_T#GREEN_LAMP:
        _TRANSIT := FALSE;
        STAMPGREENLAMP := TRUE;
        INTERCONNECTSTAMPSTARTCOMMAND := FALSE;
        IF TRUE THEN
            _TRANSIT := TRUE;
            _STATE := STAMP_STATES_T#STAMP_INIT_1;
        END_IF;

    STAMP_STATES_T#INIT:
        _TRANSIT := FALSE;
        IF TRUE THEN
            _TRANSIT := TRUE;
            _STATE := STAMP_STATES_T#START_STAMP;
        END_IF;

    STAMP_STATES_T#INTERSTEP:
        _TRANSIT := FALSE;
        STARTCOMMANDSTAMP := TRUE;
        IF STARTVAR THEN
            _TRANSIT := TRUE;
            _STATE := STAMP_STATES_T#INTERSTEP_2;
        END_IF;

    STAMP_STATES_T#INTERSTEP_2:
        _TRANSIT := FALSE;
        IF STAMPSLIDERFILLED THEN
            _TRANSIT := TRUE;
            _STATE := STAMP_STATES_T#STEP0;
        END_IF;

    STAMP_STATES_T#STAMPPROCESS:
        _TRANSIT := FALSE;
        STAMPSLIDERMOVEDIN := FALSE;
        STAMPPUSHER := TRUE;
        IF STAMPLOWERED THEN
            _TRANSIT := TRUE;
            _STATE := STAMP_STATES_T#STEP1;
        END_IF;

    STAMP_STATES_T#STAMPSLIDERBACK:
        _TRANSIT := FALSE;
        STAMPSLIDERMOVEDIN := TRUE;
        STAMPSLIDERMOVEDOUT := FALSE;
        IF STAMPSLIDERSENSORMOVEDIN THEN
            _TRANSIT := TRUE;
            _STATE := STAMP_STATES_T#STAMPPROCESS;
        END_IF;

    STAMP_STATES_T#STAMPSLIDERFORWARD:
        _TRANSIT := FALSE;
        STAMPPUSHER := FALSE;
        STAMPSLIDERMOVEDOUT := TRUE;
        IF ((STAMPLOWERED = FALSE) AND (STAMPUP = TRUE)) THEN
            INTERCONNECT := FALSE;
        END_IF;
        TIMER(IN := FALSE, PT := TIME#1MS);
        IF STAMPSLIDERMOVEDOUT THEN
            _TRANSIT := TRUE;
            _STATE := STAMP_STATES_T#STEP2;
        END_IF;

    STAMP_STATES_T#STAMP_INIT_1:
        _TRANSIT := FALSE;
        STAMPSLIDERMOVEDIN := TRUE;
        STAMPSLIDERMOVEDOUT := FALSE;
        IF STAMPSLIDERSENSORMOVEDIN THEN
            _TRANSIT := TRUE;
            _STATE := STAMP_STATES_T#STAMP_INIT_2;
        END_IF;

    STAMP_STATES_T#STAMP_INIT_2:
        _TRANSIT := FALSE;
        STAMPSLIDERMOVEDIN := FALSE;
        STAMPSLIDERMOVEDOUT := TRUE;
        IF STAMPSLIDERSENSORMOVEDOUT THEN
            _TRANSIT := TRUE;
            _STATE := STAMP_STATES_T#STAMP_INIT_3;
        END_IF;

    STAMP_STATES_T#STAMP_INIT_3:
        _TRANSIT := FALSE;
        STAMPPUSHER := TRUE;
        IF STAMPLOWERED THEN
            _TRANSIT := TRUE;
            _STATE := STAMP_STATES_T#STAMP_INIT_4;
        END_IF;

    STAMP_STATES_T#STAMP_INIT_4:
        _TRANSIT := FALSE;
        STAMPPUSHER := FALSE;
        IF STAMPUP THEN
            _TRANSIT := TRUE;
            _STATE := STAMP_STATES_T#INTERSTEP;
        END_IF;

    STAMP_STATES_T#START_STAMP:
        _TRANSIT := FALSE;
        STAMPSLIDERMOVEDOUT := FALSE;
        STAMPSLIDERMOVEDIN := FALSE;
        STAMPPUSHER := FALSE;
        STAMPGREENLAMP := FALSE;
        STAMPPRESSURE := FALSE;
        STARTCOMMANDSTAMP := FALSE;
        IF (STAMPSTARTBUTTON = TRUE) THEN
            INTERCONNECTSTAMPSTARTCOMMAND := TRUE;
        END_IF;
        IF INTERCONNECTSTAMPSTARTCOMMAND THEN
            _TRANSIT := TRUE;
            _STATE := STAMP_STATES_T#GREEN_LAMP;
        END_IF;

    STAMP_STATES_T#STEP0:
        _TRANSIT := FALSE;
        IF CRANEUP THEN
            _TRANSIT := TRUE;
            _STATE := STAMP_STATES_T#STAMPSLIDERBACK;
        END_IF;

    STAMP_STATES_T#STEP1:
        _TRANSIT := FALSE;
        TIMER(IN := STAMPLOWERED, PT := TIME#12ms);
        INTERCONNECT := TIMER.Q;
        IF INTERCONNECT THEN
            _TRANSIT := TRUE;
            _STATE := STAMP_STATES_T#STAMPSLIDERFORWARD;
        END_IF;

    STAMP_STATES_T#STEP2:
        _TRANSIT := FALSE;
        IF (CRANEONCONVEYOR AND NOT STAMPSLIDERFILLED) THEN
            _TRANSIT := TRUE;
            _STATE := STAMP_STATES_T#INTERSTEP;
        END_IF;

    END_CASE;
END_FUNCTION_BLOCK

FUNCTION_BLOCK CRANE_FB
VAR_OUTPUT  ANALOGCRANEPRESSURE : INT; END_VAR
VAR_INPUT  CRANEDOWN : BOOL; END_VAR
VAR_OUTPUT  CRANELOWER : BOOL; END_VAR
VAR_INPUT  CRANEONCONVEYOR : BOOL; END_VAR
VAR_INPUT  CRANEONMAGAZIN : BOOL; END_VAR
VAR_INPUT  CRANEPOSITIONSTAMP : BOOL; END_VAR
VAR_INPUT  CRANESUCKED : BOOL; END_VAR
VAR_OUTPUT  CRANETURNCLOCKWISE : BOOL; END_VAR
VAR_OUTPUT  CRANETURNCOUNTERCLOCKWISE : BOOL; END_VAR
VAR_INPUT  CRANEUP : BOOL; END_VAR
VAR  DURATION1 : TIME := TIME#1S500MS; END_VAR
VAR_INPUT  MAGAZINCAPACITIVESENSOR : BOOL; END_VAR
VAR_INPUT  MAGAZINOPTICALSENSOR : BOOL; END_VAR
VAR_OUTPUT  MAGAZINVACUUMOFF : BOOL; END_VAR
VAR_OUTPUT  MAGAZINVACUUMON : BOOL; END_VAR
VAR  SFCINIT : BOOL; END_VAR
VAR_INPUT  SFCRESET : BOOL; END_VAR
VAR_INPUT  SLIDERMOVEDOUT : BOOL; END_VAR
VAR_INPUT  SLIDERNOTMOVEDOUT : BOOL; END_VAR
VAR_INPUT  STAMPLOWERED : BOOL; END_VAR
VAR_INPUT  STAMPSLIDERFILLED : BOOL; END_VAR
VAR_INPUT  STAMPSLIDERSENSORMOVEDOUT : BOOL; END_VAR
VAR_INPUT  STARTBUTTONMAGAZIN : BOOL; END_VAR
VAR_OUTPUT  STARTCOMMANDCRANE : BOOL; END_VAR
VAR_INPUT  STARTVAR : BOOL; END_VAR
VAR  TIMEDELAY_TIMER : TON; END_VAR
VAR  TIMEDELAY_TIMER_DURATION : TIME := TIME#50MS; END_VAR
VAR  TIMEDELAY_TIMER_INTERCONNECT : BOOL; END_VAR
VAR  TIMER1 : TON; END_VAR
VAR_INPUT  WORKPIECEREADY : BOOL; END_VAR
VAR  _STATE : CRANE_STATES_T; END_VAR
VAR  _TRANSIT : BOOL; END_VAR
VAR  ACTUALTIME1 : TIME; END_VAR
VAR  INTERCONNECT : BOOL; END_VAR
VAR  INTERCONNECTCRANESTARTCOMMAND : BOOL; END_VAR

CASE _STATE OF
    CRANE_STATES_T#CRANE_GO_UP:
        _TRANSIT := FALSE;
        CRANELOWER := FALSE;
        IF CRANEUP THEN
            _TRANSIT := TRUE;
            _STATE := CRANE_STATES_T#STEP3;
        END_IF;

    CRANE_STATES_T#CRANE_GO_UP_WHITE:
        _TRANSIT := FALSE;
        CRANELOWER := FALSE;
        IF CRANEUP THEN
            _TRANSIT := TRUE;
            _STATE := CRANE_STATES_T#STEP3;
        END_IF;

    CRANE_STATES_T#CRANE_INIT:
        _TRANSIT := FALSE;
        CRANELOWER := TRUE;
        INTERCONNECTCRANESTARTCOMMAND := FALSE;
        ANALOGCRANEPRESSURE := INT#6000;
        IF CRANEDOWN THEN
            _TRANSIT := TRUE;
            _STATE := CRANE_STATES_T#CRANE_INIT_2;
        END_IF;

    CRANE_STATES_T#CRANE_INIT_2:
        _TRANSIT := FALSE;
        CRANELOWER := FALSE;
        IF CRANEUP THEN
            _TRANSIT := TRUE;
            _STATE := CRANE_STATES_T#INTERSTEP;
        END_IF;

    CRANE_STATES_T#CRANE_LIFT_AT_STAMP:
        _TRANSIT := FALSE;
        CRANELOWER := FALSE;
        IF CRANEUP THEN
            _TRANSIT := TRUE;
            _STATE := CRANE_STATES_T#CRANE_TURN_LEFT_FROM_STAMP;
        END_IF;

    CRANE_STATES_T#CRANE_LIFT_AT_STAMP2:
        _TRANSIT := FALSE;
        CRANELOWER := FALSE;
        IF CRANEUP THEN
            _TRANSIT := TRUE;
            _STATE := CRANE_STATES_T#CRANE_TURN_RIGHT_FROM_STAMP;
        END_IF;

    CRANE_STATES_T#CRANE_LIFT_CONVEYOR:
        _TRANSIT := FALSE;
        CRANELOWER := FALSE;
        IF TRUE THEN
            _TRANSIT := TRUE;
            _STATE := CRANE_STATES_T#INTERSTEP;
        END_IF;

    CRANE_STATES_T#CRANE_LIFT_CONVEYOR2:
        _TRANSIT := FALSE;
        CRANELOWER := FALSE;
        IF TRUE THEN
            _TRANSIT := TRUE;
            _STATE := CRANE_STATES_T#INTERSTEP;
        END_IF;

    CRANE_STATES_T#CRANE_LIFT_CONVEYOR_BLACK:
        _TRANSIT := FALSE;
        CRANELOWER := FALSE;
        IF CRANEUP THEN
            _TRANSIT := TRUE;
            _STATE := CRANE_STATES_T#CRANE_TURN_LEFT_BACK_TO_STAMP;
        END_IF;

    CRANE_STATES_T#CRANE_LIFT_MAGAZIN:
        _TRANSIT := FALSE;
        CRANELOWER := FALSE;
        IF CRANEUP THEN
            _TRANSIT := TRUE;
            _STATE := CRANE_STATES_T#CRANE_TURN_LEFT_NOT_METALLIC;
        END_IF;

    CRANE_STATES_T#CRANE_LIFT_MAGAZIN_METALLIC:
        _TRANSIT := FALSE;
        CRANELOWER := FALSE;
        IF CRANEUP THEN
            _TRANSIT := TRUE;
            _STATE := CRANE_STATES_T#CRANE_TURN_LEFT_METALLIC;
        END_IF;

    CRANE_STATES_T#CRANE_LIFT_MAGAZINE_WHITE:
        _TRANSIT := FALSE;
        CRANELOWER := FALSE;
        IF CRANEUP THEN
            _TRANSIT := TRUE;
            _STATE := CRANE_STATES_T#CRANE_TURN_LEFT_WHITE;
        END_IF;

    CRANE_STATES_T#CRANE_LIFT_NOT_METALLIC_BLACK:
        _TRANSIT := FALSE;
        CRANELOWER := FALSE;
        IF CRANEUP THEN
            _TRANSIT := TRUE;
            _STATE := CRANE_STATES_T#CRANE_TURN_LEFT_NOT_METALLIC_BLACK;
        END_IF;

    CRANE_STATES_T#CRANE_LOWER:
        _TRANSIT := FALSE;
        MAGAZINVACUUMON := TRUE;
        MAGAZINVACUUMOFF := FALSE;
        CRANELOWER := TRUE;
        ANALOGCRANEPRESSURE := INT#0;
        IF CRANESUCKED THEN
            _TRANSIT := TRUE;
            _STATE := CRANE_STATES_T#STEP0;
        END_IF;

    CRANE_STATES_T#CRANE_ON_CONVEYOR:
        _TRANSIT := FALSE;
        CRANETURNCOUNTERCLOCKWISE := FALSE;
        CRANETURNCLOCKWISE := FALSE;
        CRANELOWER := TRUE;
        IF CRANEDOWN THEN
            _TRANSIT := TRUE;
            _STATE := CRANE_STATES_T#RELEASE;
        END_IF;

    CRANE_STATES_T#CRANE_ON_CONVEYOR_METALLIC:
        _TRANSIT := FALSE;
        CRANETURNCOUNTERCLOCKWISE := FALSE;
        CRANETURNCLOCKWISE := FALSE;
        CRANELOWER := TRUE;
        IF CRANEDOWN THEN
            _TRANSIT := TRUE;
            _STATE := CRANE_STATES_T#RELEASE;
        END_IF;

    CRANE_STATES_T#CRANE_ON_CONVEYOR_METALLIC2:
        _TRANSIT := FALSE;
        CRANETURNCOUNTERCLOCKWISE := FALSE;
        CRANETURNCLOCKWISE := FALSE;
        CRANELOWER := TRUE;
        IF CRANEDOWN THEN
            _TRANSIT := TRUE;
            _STATE := CRANE_STATES_T#RELEASE2;
        END_IF;

    CRANE_STATES_T#CRANE_ON_CONVEYOR_NOT_METALLICA_BLACK:
        _TRANSIT := FALSE;
        CRANETURNCOUNTERCLOCKWISE := FALSE;
        CRANETURNCLOCKWISE := FALSE;
        CRANELOWER := TRUE;
        IF CRANEDOWN THEN
            _TRANSIT := TRUE;
            _STATE := CRANE_STATES_T#RELEASE_BLACK;
        END_IF;

    CRANE_STATES_T#CRANE_ON_STAMP_METALLIC:
        _TRANSIT := FALSE;
        CRANETURNCOUNTERCLOCKWISE := FALSE;
        CRANETURNCLOCKWISE := FALSE;
        CRANELOWER := TRUE;
        IF CRANEDOWN THEN
            _TRANSIT := TRUE;
            _STATE := CRANE_STATES_T#RELEASE_WORKPIECE;
        END_IF;

    CRANE_STATES_T#CRANE_ON_STAMP_METALLIC2:
        _TRANSIT := FALSE;
        CRANETURNCOUNTERCLOCKWISE := FALSE;
        CRANETURNCLOCKWISE := FALSE;
        IF STAMPLOWERED THEN
            _TRANSIT := TRUE;
            _STATE := CRANE_STATES_T#INTERSTEP_4;
        END_IF;

    CRANE_STATES_T#CRANE_ON_STAMP_METALLIC2_LOWER:
        _TRANSIT := FALSE;
        CRANELOWER := TRUE;
        IF CRANEDOWN THEN
            _TRANSIT := TRUE;
            _STATE := CRANE_STATES_T#SUCK_AT_STAMP2;
        END_IF;

    CRANE_STATES_T#CRANE_ON_STAMP_STOP_BLACK:
        _TRANSIT := FALSE;
        CRANETURNCLOCKWISE := FALSE;
        CRANETURNCOUNTERCLOCKWISE := FALSE;
        IF TRUE THEN
            _TRANSIT := TRUE;
            _STATE := CRANE_STATES_T#RESET_INTERCONNECT;
        END_IF;

    CRANE_STATES_T#CRANE_ON_STAMP_WHITE:
        _TRANSIT := FALSE;
        CRANETURNCOUNTERCLOCKWISE := FALSE;
        CRANETURNCLOCKWISE := FALSE;
        CRANELOWER := TRUE;
        IF CRANEDOWN THEN
            _TRANSIT := TRUE;
            _STATE := CRANE_STATES_T#RELEASE_WORKPIECE_WHITE;
        END_IF;

    CRANE_STATES_T#CRANE_TURN_LEFT_BACK_TO_STAMP:
        _TRANSIT := FALSE;
        CRANETURNCOUNTERCLOCKWISE := TRUE;
        CRANETURNCLOCKWISE := FALSE;
        IF CRANEPOSITIONSTAMP THEN
            _TRANSIT := TRUE;
            _STATE := CRANE_STATES_T#CRANE_ON_STAMP_STOP_BLACK;
        END_IF;

    CRANE_STATES_T#CRANE_TURN_LEFT_FROM_STAMP:
        _TRANSIT := FALSE;
        CRANETURNCLOCKWISE := TRUE;
        CRANETURNCOUNTERCLOCKWISE := FALSE;
        IF CRANEONCONVEYOR THEN
            _TRANSIT := TRUE;
            _STATE := CRANE_STATES_T#CRANE_ON_CONVEYOR_METALLIC;
        END_IF;

    CRANE_STATES_T#CRANE_TURN_LEFT_METALLIC:
        _TRANSIT := FALSE;
        CRANETURNCOUNTERCLOCKWISE := TRUE;
        CRANETURNCLOCKWISE := FALSE;
        IF CRANEPOSITIONSTAMP THEN
            _TRANSIT := TRUE;
            _STATE := CRANE_STATES_T#CRANE_ON_STAMP_METALLIC;
        END_IF;

    CRANE_STATES_T#CRANE_TURN_LEFT_METALLIC2:
        _TRANSIT := FALSE;
        CRANETURNCOUNTERCLOCKWISE := TRUE;
        CRANETURNCLOCKWISE := FALSE;
        IF CRANEPOSITIONSTAMP THEN
            _TRANSIT := TRUE;
            _STATE := CRANE_STATES_T#CRANE_ON_STAMP_METALLIC2;
        END_IF;

    CRANE_STATES_T#CRANE_TURN_LEFT_NOT_METALLIC:
        _TRANSIT := FALSE;
        CRANETURNCOUNTERCLOCKWISE := TRUE;
        CRANETURNCLOCKWISE := FALSE;
        IF CRANEONCONVEYOR THEN
            _TRANSIT := TRUE;
            _STATE := CRANE_STATES_T#CRANE_ON_CONVEYOR;
        END_IF;

    CRANE_STATES_T#CRANE_TURN_LEFT_NOT_METALLIC_BLACK:
        _TRANSIT := FALSE;
        CRANETURNCOUNTERCLOCKWISE := TRUE;
        CRANETURNCLOCKWISE := FALSE;
        IF CRANEONCONVEYOR THEN
            _TRANSIT := TRUE;
            _STATE := CRANE_STATES_T#CRANE_ON_CONVEYOR_NOT_METALLICA_BLACK;
        END_IF;

    CRANE_STATES_T#CRANE_TURN_LEFT_WHITE:
        _TRANSIT := FALSE;
        CRANETURNCOUNTERCLOCKWISE := TRUE;
        CRANETURNCLOCKWISE := FALSE;
        IF CRANEPOSITIONSTAMP THEN
            _TRANSIT := TRUE;
            _STATE := CRANE_STATES_T#CRANE_ON_STAMP_WHITE;
        END_IF;

    CRANE_STATES_T#CRANE_TURN_RIGHT_FROM_STAMP:
        _TRANSIT := FALSE;
        CRANETURNCLOCKWISE := TRUE;
        CRANETURNCOUNTERCLOCKWISE := FALSE;
        IF CRANEONCONVEYOR THEN
            _TRANSIT := TRUE;
            _STATE := CRANE_STATES_T#CRANE_ON_CONVEYOR_METALLIC2;
        END_IF;

    CRANE_STATES_T#INIT:
        _TRANSIT := FALSE;
        IF TRUE THEN
            _TRANSIT := TRUE;
            _STATE := CRANE_STATES_T#START_CRANE;
        END_IF;

    CRANE_STATES_T#INTERSTEP:
        _TRANSIT := FALSE;
        STARTCOMMANDCRANE := TRUE;
        IF STARTVAR THEN
            _TRANSIT := TRUE;
            _STATE := CRANE_STATES_T#INTERSTEP_2;
        END_IF;

    CRANE_STATES_T#INTERSTEP_2:
        _TRANSIT := FALSE;
        IF SLIDERMOVEDOUT THEN
            _TRANSIT := TRUE;
            _STATE := CRANE_STATES_T#TIMEDELAY;
        END_IF;

    CRANE_STATES_T#INTERSTEP_3:
        _TRANSIT := FALSE;
        IF NOT WORKPIECEREADY THEN
            _TRANSIT := TRUE;
            _STATE := CRANE_STATES_T#NO_WORKPIECE_READY;
        ELSIF WORKPIECEREADY THEN
            _TRANSIT := TRUE;
            _STATE := CRANE_STATES_T#TURN_RIGHT;
        END_IF;

    CRANE_STATES_T#INTERSTEP_4:
        _TRANSIT := FALSE;
        IF STAMPSLIDERSENSORMOVEDOUT THEN
            _TRANSIT := TRUE;
            _STATE := CRANE_STATES_T#CRANE_ON_STAMP_METALLIC2_LOWER;
        END_IF;

    CRANE_STATES_T#LOWER_CRANE:
        _TRANSIT := FALSE;
        CRANELOWER := TRUE;
        IF CRANEDOWN THEN
            _TRANSIT := TRUE;
            _STATE := CRANE_STATES_T#SUCK_AT_STAMP;
        END_IF;

    CRANE_STATES_T#MAGAZIN_STOP:
        _TRANSIT := FALSE;
        CRANETURNCLOCKWISE := FALSE;
        CRANETURNCOUNTERCLOCKWISE := FALSE;
        IF TRUE THEN
            _TRANSIT := TRUE;
            _STATE := CRANE_STATES_T#CRANE_LOWER;
        END_IF;

    CRANE_STATES_T#MAGAZIN_STOP_BLACK:
        _TRANSIT := FALSE;
        CRANETURNCLOCKWISE := FALSE;
        CRANETURNCOUNTERCLOCKWISE := FALSE;
        MAGAZINVACUUMON := TRUE;
        MAGAZINVACUUMOFF := FALSE;
        CRANELOWER := TRUE;
        IF CRANESUCKED THEN
            _TRANSIT := TRUE;
            _STATE := CRANE_STATES_T#CRANE_LIFT_NOT_METALLIC_BLACK;
        END_IF;

    CRANE_STATES_T#MAGAZIN_STOP_FINAL:
        _TRANSIT := FALSE;
        CRANETURNCLOCKWISE := FALSE;
        CRANETURNCOUNTERCLOCKWISE := FALSE;
        IF TRUE THEN
            _TRANSIT := TRUE;
            _STATE := CRANE_STATES_T#START_CRANE;
        END_IF;

    CRANE_STATES_T#NO_WORKPIECE_READY:
        _TRANSIT := FALSE;
        MAGAZINVACUUMON := FALSE;
        MAGAZINVACUUMOFF := FALSE;
        CRANELOWER := FALSE;
        IF NOT STAMPSLIDERFILLED THEN
            _TRANSIT := TRUE;
            _STATE := CRANE_STATES_T#TURN_RIGHT_FINAL;
        ELSIF STAMPSLIDERFILLED THEN
            _TRANSIT := TRUE;
            _STATE := CRANE_STATES_T#CRANE_TURN_LEFT_METALLIC2;
        END_IF;

    CRANE_STATES_T#RESET_INTERCONNECT:
        _TRANSIT := FALSE;
        INTERCONNECT := FALSE;
        TIMER1(IN := FALSE, PT := TIME#1MS);
        IF SLIDERMOVEDOUT THEN
            _TRANSIT := TRUE;
            _STATE := CRANE_STATES_T#LOWER_CRANE;
        END_IF;

    CRANE_STATES_T#STAMP_PRESSURE_PROFILE_SET_METALLIC:
        _TRANSIT := FALSE;
        ANALOGCRANEPRESSURE := INT#7000;
        IF TRUE THEN
            _TRANSIT := TRUE;
            _STATE := CRANE_STATES_T#CRANE_LIFT_MAGAZIN_METALLIC;
        END_IF;

    CRANE_STATES_T#STAMP_PRESSURE_PROFILE_SET_WHITE:
        _TRANSIT := FALSE;
        ANALOGCRANEPRESSURE := INT#6000;
        IF TRUE THEN
            _TRANSIT := TRUE;
            _STATE := CRANE_STATES_T#CRANE_LIFT_MAGAZINE_WHITE;
        END_IF;

    CRANE_STATES_T#START_CRANE:
        _TRANSIT := FALSE;
        CRANELOWER := FALSE;
        MAGAZINVACUUMOFF := TRUE;
        MAGAZINVACUUMON := FALSE;
        CRANETURNCOUNTERCLOCKWISE := FALSE;
        CRANETURNCLOCKWISE := FALSE;
        STARTVAR := FALSE;
        STARTCOMMANDCRANE := FALSE;
        IF (STARTBUTTONMAGAZIN = TRUE) THEN
            INTERCONNECTCRANESTARTCOMMAND := TRUE;
        END_IF;
        IF INTERCONNECTCRANESTARTCOMMAND THEN
            _TRANSIT := TRUE;
            _STATE := CRANE_STATES_T#CRANE_INIT;
        END_IF;

    CRANE_STATES_T#STEP0:
        _TRANSIT := FALSE;
        IF (NOT MAGAZINCAPACITIVESENSOR AND MAGAZINOPTICALSENSOR) THEN
            _TRANSIT := TRUE;
            _STATE := CRANE_STATES_T#STAMP_PRESSURE_PROFILE_SET_WHITE;
        ELSIF (MAGAZINCAPACITIVESENSOR AND MAGAZINOPTICALSENSOR) THEN
            _TRANSIT := TRUE;
            _STATE := CRANE_STATES_T#STAMP_PRESSURE_PROFILE_SET_METALLIC;
        ELSIF (NOT MAGAZINCAPACITIVESENSOR AND NOT MAGAZINOPTICALSENSOR) THEN
            _TRANSIT := TRUE;
            _STATE := CRANE_STATES_T#CRANE_LIFT_MAGAZIN;
        END_IF;

    CRANE_STATES_T#STEP2:
        _TRANSIT := FALSE;
        IF (MAGAZINCAPACITIVESENSOR OR MAGAZINOPTICALSENSOR) THEN
            _TRANSIT := TRUE;
            _STATE := CRANE_STATES_T#PAUSE;
        ELSIF (NOT MAGAZINCAPACITIVESENSOR AND NOT MAGAZINOPTICALSENSOR) THEN
            _TRANSIT := TRUE;
            _STATE := CRANE_STATES_T#TURN_RIGHT_BLACK;
        END_IF;

    CRANE_STATES_T#STEP3:
        _TRANSIT := FALSE;
        IF NOT WORKPIECEREADY THEN
            _TRANSIT := TRUE;
            _STATE := CRANE_STATES_T#STEP4;
        ELSIF WORKPIECEREADY THEN
            _TRANSIT := TRUE;
            _STATE := CRANE_STATES_T#STEP2;
        END_IF;

    CRANE_STATES_T#STEP4:
        _TRANSIT := FALSE;
        IF TRUE THEN
            _TRANSIT := TRUE;
            _STATE := CRANE_STATES_T#INTERSTEP;
        END_IF;

    CRANE_STATES_T#SUCK_AT_STAMP:
        _TRANSIT := FALSE;
        MAGAZINVACUUMON := TRUE;
        MAGAZINVACUUMOFF := FALSE;
        IF CRANESUCKED THEN
            _TRANSIT := TRUE;
            _STATE := CRANE_STATES_T#CRANE_LIFT_AT_STAMP;
        END_IF;

    CRANE_STATES_T#SUCK_AT_STAMP2:
        _TRANSIT := FALSE;
        MAGAZINVACUUMON := TRUE;
        MAGAZINVACUUMOFF := FALSE;
        IF CRANESUCKED THEN
            _TRANSIT := TRUE;
            _STATE := CRANE_STATES_T#CRANE_LIFT_AT_STAMP2;
        END_IF;

    CRANE_STATES_T#TIMEDELAY:
        _TRANSIT := FALSE;
        TIMEDELAY_TIMER(IN := TRUE, PT := TIMEDELAY_TIMER_DURATION);
        TIMEDELAY_TIMER_INTERCONNECT := TIMEDELAY_TIMER.Q;
        IF TIMEDELAY_TIMER_INTERCONNECT THEN
            _TRANSIT := TRUE;
            _STATE := CRANE_STATES_T#INTERSTEP_3;
        END_IF;

    CRANE_STATES_T#TURN_RIGHT:
        _TRANSIT := FALSE;
        CRANETURNCLOCKWISE := TRUE;
        CRANETURNCOUNTERCLOCKWISE := FALSE;
        IF CRANEONMAGAZIN THEN
            _TRANSIT := TRUE;
            _STATE := CRANE_STATES_T#MAGAZIN_STOP;
        END_IF;

    CRANE_STATES_T#TURN_RIGHT_BLACK:
        _TRANSIT := FALSE;
        CRANETURNCLOCKWISE := TRUE;
        CRANETURNCOUNTERCLOCKWISE := FALSE;
        IF CRANEONMAGAZIN THEN
            _TRANSIT := TRUE;
            _STATE := CRANE_STATES_T#MAGAZIN_STOP_BLACK;
        END_IF;

    CRANE_STATES_T#TURN_RIGHT_FINAL:
        _TRANSIT := FALSE;
        CRANETURNCLOCKWISE := TRUE;
        CRANETURNCOUNTERCLOCKWISE := FALSE;
        ANALOGCRANEPRESSURE := INT#0;
        IF CRANEONMAGAZIN THEN
            _TRANSIT := TRUE;
            _STATE := CRANE_STATES_T#MAGAZIN_STOP_FINAL;
        END_IF;

    CRANE_STATES_T#PAUSE:
        _TRANSIT := FALSE;
        TIMER1(IN := CRANEUP, PT := DURATION1);
        INTERCONNECT := TIMER1.Q;
        IF INTERCONNECT THEN
            _TRANSIT := TRUE;
            _STATE := CRANE_STATES_T#RESET_INTERCONNECT;
        END_IF;

    CRANE_STATES_T#RELEASE:
        _TRANSIT := FALSE;
        MAGAZINVACUUMOFF := TRUE;
        MAGAZINVACUUMON := FALSE;
        IF TRUE THEN
            _TRANSIT := TRUE;
            _STATE := CRANE_STATES_T#CRANE_LIFT_CONVEYOR;
        END_IF;

    CRANE_STATES_T#RELEASE2:
        _TRANSIT := FALSE;
        MAGAZINVACUUMOFF := TRUE;
        MAGAZINVACUUMON := FALSE;
        IF TRUE THEN
            _TRANSIT := TRUE;
            _STATE := CRANE_STATES_T#CRANE_LIFT_CONVEYOR2;
        END_IF;

    CRANE_STATES_T#RELEASE_BLACK:
        _TRANSIT := FALSE;
        MAGAZINVACUUMON := FALSE;
        MAGAZINVACUUMOFF := TRUE;
        IF TRUE THEN
            _TRANSIT := TRUE;
            _STATE := CRANE_STATES_T#CRANE_LIFT_CONVEYOR_BLACK;
        END_IF;

    CRANE_STATES_T#RELEASE_WORKPIECE:
        _TRANSIT := FALSE;
        MAGAZINVACUUMOFF := TRUE;
        MAGAZINVACUUMON := FALSE;
        IF TRUE THEN
            _TRANSIT := TRUE;
            _STATE := CRANE_STATES_T#CRANE_GO_UP;
        END_IF;

    CRANE_STATES_T#RELEASE_WORKPIECE_WHITE:
        _TRANSIT := FALSE;
        MAGAZINVACUUMOFF := TRUE;
        MAGAZINVACUUMON := FALSE;
        IF TRUE THEN
            _TRANSIT := TRUE;
            _STATE := CRANE_STATES_T#CRANE_GO_UP_WHITE;
        END_IF;

    END_CASE;
END_FUNCTION_BLOCK

PROGRAM MAIN

VAR  ACTUATOR_ANALOGCRANEPRESSURE : INT; END_VAR
VAR  ACTUATOR_CRANELOWER : BOOL; END_VAR
VAR  ACTUATOR_CRANETURNCLOCKWISE : BOOL; END_VAR
VAR  ACTUATOR_CRANETURNCOUNTERCLOCKWISE : BOOL; END_VAR
VAR  ACTUATOR_MAGAZINGREENLAMP : BOOL; END_VAR
VAR  ACTUATOR_MAGAZINSLIDER : BOOL; END_VAR
VAR  ACTUATOR_MAGAZINVACUUMOFF : BOOL; END_VAR
VAR  ACTUATOR_MAGAZINVACUUMON : BOOL; END_VAR
VAR  ACTUATOR_MAGAZINWHITELAMP : BOOL; END_VAR
VAR  ACTUATOR_STAMPGREENLAMP : BOOL; END_VAR
VAR  ACTUATOR_STAMPPUSHER : BOOL; END_VAR
VAR  ACTUATOR_STAMPSLIDERMOVEDIN : BOOL; END_VAR
VAR  ACTUATOR_STAMPSLIDERMOVEDOUT : BOOL; END_VAR
VAR  ACTUATOR_STAMPWHITELAMP : BOOL; END_VAR
VAR  CRANE : CRANE_FB; END_VAR
VAR  MAG : MAGAZIN; END_VAR
VAR  SENSOR_CRANEDOWN : BOOL; END_VAR
VAR  SENSOR_CRANEONCONVEYOR : BOOL; END_VAR
VAR  SENSOR_CRANEONMAGAZIN : BOOL; END_VAR
VAR  SENSOR_CRANEPOSITION : BOOL; END_VAR
VAR  SENSOR_CRANEPOSITIONSTAMP : BOOL; END_VAR
VAR  SENSOR_CRANESUCKED : BOOL; END_VAR
VAR  SENSOR_CRANEUP : BOOL; END_VAR
VAR  SENSOR_MAGAZINCAPACITIVESENSOR : BOOL; END_VAR
VAR  SENSOR_MAGAZINEMERGENCYSTOP : BOOL; END_VAR
VAR  SENSOR_MAGAZINOPTICALSENSOR : BOOL; END_VAR
VAR  SENSOR_MAGAZINSWITCHMANUELLAUTOMATIC : BOOL; END_VAR
VAR  SENSOR_SLIDERMOVEDOUT : BOOL; END_VAR
VAR  SENSOR_SLIDERNOTMOVEDOUT : BOOL; END_VAR
VAR  SENSOR_STAMPEMERGENCYSTOP : BOOL; END_VAR
VAR  SENSOR_STAMPLOWERED : BOOL; END_VAR
VAR  SENSOR_STAMPSLIDERFILLED : BOOL; END_VAR
VAR  SENSOR_STAMPSLIDERSENSORMOVEDIN : BOOL; END_VAR
VAR  SENSOR_STAMPSLIDERSENSORMOVEDOUT : BOOL; END_VAR
VAR  SENSOR_STAMPSTARTBUTTON : BOOL; END_VAR
VAR  SENSOR_STAMPSWITCHMANUELLAUTOMATIC : BOOL; END_VAR
VAR  SENSOR_STAMPUP : BOOL; END_VAR
VAR  SENSOR_STARTBUTTONMAGAZIN : BOOL; END_VAR
VAR  SENSOR_WORKPIECEREADY : BOOL; END_VAR
VAR  STAMP : STAMP_FB; END_VAR
MAG.SLIDERNOTMOVEDOUT := SENSOR_SLIDERNOTMOVEDOUT;
MAG.SLIDERMOVEDOUT := SENSOR_SLIDERMOVEDOUT;
MAG.CRANEONMAGAZIN := SENSOR_CRANEONMAGAZIN;
MAG.CRANEDOWN := SENSOR_CRANEDOWN;
MAG.CRANEUP := SENSOR_CRANEUP;
MAG.CRANEONCONVEYOR := SENSOR_CRANEONCONVEYOR;
MAG.WORKPIECEREADY := SENSOR_WORKPIECEREADY;
MAG.STARTBUTTONMAGAZIN := SENSOR_STARTBUTTONMAGAZIN;
ACTUATOR_MAGAZINSLIDER := MAG.MAGAZINSLIDER;
ACTUATOR_MAGAZINGREENLAMP := MAG.MAGAZINGREENLAMP;
CRANE.CRANEUP := SENSOR_CRANEUP;
CRANE.CRANEONCONVEYOR := SENSOR_CRANEONCONVEYOR;
CRANE.CRANEDOWN := SENSOR_CRANEDOWN;
CRANE.CRANESUCKED := SENSOR_CRANESUCKED;
CRANE.CRANEONMAGAZIN := SENSOR_CRANEONMAGAZIN;
CRANE.MAGAZINCAPACITIVESENSOR := SENSOR_MAGAZINCAPACITIVESENSOR;
CRANE.CRANEPOSITIONSTAMP := SENSOR_CRANEPOSITIONSTAMP;
CRANE.SLIDERMOVEDOUT := SENSOR_SLIDERMOVEDOUT;
CRANE.WORKPIECEREADY := SENSOR_WORKPIECEREADY;
CRANE.MAGAZINOPTICALSENSOR := SENSOR_MAGAZINOPTICALSENSOR;
CRANE.STAMPSLIDERFILLED := SENSOR_STAMPSLIDERFILLED;
CRANE.STAMPSLIDERSENSORMOVEDOUT := SENSOR_STAMPSLIDERSENSORMOVEDOUT;
CRANE.STAMPLOWERED := SENSOR_STAMPLOWERED;
CRANE.STARTBUTTONMAGAZIN := SENSOR_STARTBUTTONMAGAZIN;
ACTUATOR_CRANETURNCOUNTERCLOCKWISE := CRANE.CRANETURNCOUNTERCLOCKWISE;
ACTUATOR_CRANETURNCLOCKWISE := CRANE.CRANETURNCLOCKWISE;
ACTUATOR_CRANELOWER := CRANE.CRANELOWER;
ACTUATOR_MAGAZINVACUUMOFF := CRANE.MAGAZINVACUUMOFF;
ACTUATOR_MAGAZINVACUUMON := CRANE.MAGAZINVACUUMON;
ACTUATOR_ANALOGCRANEPRESSURE := CRANE.ANALOGCRANEPRESSURE;
STAMP.STAMPSLIDERSENSORMOVEDOUT := SENSOR_STAMPSLIDERSENSORMOVEDOUT;
STAMP.STAMPSLIDERSENSORMOVEDIN := SENSOR_STAMPSLIDERSENSORMOVEDIN;
STAMP.STAMPSLIDERFILLED := SENSOR_STAMPSLIDERFILLED;
STAMP.STAMPUP := SENSOR_STAMPUP;
STAMP.STAMPLOWERED := SENSOR_STAMPLOWERED;
STAMP.CRANEDOWN := SENSOR_CRANEDOWN;
STAMP.CRANEUP := SENSOR_CRANEUP;
STAMP.CRANESUCKED := SENSOR_CRANESUCKED;
STAMP.CRANEPOSITIONSTAMP := SENSOR_CRANEPOSITIONSTAMP;
STAMP.CRANEONCONVEYOR := SENSOR_CRANEONCONVEYOR;
STAMP.STAMPSTARTBUTTON := SENSOR_STAMPSTARTBUTTON;
ACTUATOR_STAMPSLIDERMOVEDOUT := STAMP.STAMPSLIDERMOVEDOUT;
ACTUATOR_STAMPSLIDERMOVEDIN := STAMP.STAMPSLIDERMOVEDIN;
ACTUATOR_STAMPWHITELAMP := STAMP.STAMPWHITELAMP;
ACTUATOR_STAMPPUSHER := STAMP.STAMPPUSHER;
ACTUATOR_STAMPGREENLAMP := STAMP.STAMPGREENLAMP;
IF (SENSOR_STAMPEMERGENCYSTOP AND SENSOR_MAGAZINEMERGENCYSTOP) THEN
    MAG();
    CRANE();
    STAMP();
    IF (ACTUATOR_MAGAZINGREENLAMP AND ACTUATOR_STAMPGREENLAMP) THEN
        IF ((STAMP.STARTCOMMANDSTAMP AND CRANE.STARTCOMMANDCRANE) AND MAG.STARTCOMMANDMAGAZIN) THEN
            CRANE.STARTVAR := TRUE;
            MAG.STARTVAR := TRUE;
            STAMP.STARTVAR := TRUE;
        END_IF;
    END_IF;
    CRANE.SFCRESET := FALSE;
    MAG.SFCRESET := FALSE;
    STAMP.SFCRESET := FALSE;
ELSIF (NOT SENSOR_STAMPEMERGENCYSTOP OR NOT SENSOR_MAGAZINEMERGENCYSTOP) THEN
    ACTUATOR_MAGAZINSLIDER := FALSE;
    ACTUATOR_CRANELOWER := FALSE;
    ACTUATOR_MAGAZINVACUUMON := FALSE;
    ACTUATOR_MAGAZINVACUUMOFF := TRUE;
    ACTUATOR_MAGAZINGREENLAMP := FALSE;
    ACTUATOR_CRANETURNCOUNTERCLOCKWISE := FALSE;
    ACTUATOR_CRANETURNCLOCKWISE := FALSE;
    ACTUATOR_STAMPSLIDERMOVEDOUT := TRUE;
    ACTUATOR_STAMPSLIDERMOVEDIN := FALSE;
    ACTUATOR_STAMPGREENLAMP := FALSE;
    ACTUATOR_STAMPPUSHER := FALSE;
    ACTUATOR_ANALOGCRANEPRESSURE := INT#0;
    CRANE.SFCRESET := TRUE;
    MAG.SFCRESET := TRUE;
    STAMP.SFCRESET := TRUE;
    CRANE.STARTVAR := FALSE;
    MAG.STARTVAR := FALSE;
    STAMP.STARTVAR := FALSE;
END_IF;
END_PROGRAM

CONFIGURATION Config0
  RESOURCE Res0 ON PLC
    TASK TASK0(INTERVAL := T#50MS, PRIORITY := 0);
    PROGRAM INSTANCE0 WITH TASK0 : MAIN;
  END_RESOURCE
END_CONFIGURATION
